{attribute 'qualified_only'}
VAR_GLOBAL
END_VAR

(* stored: Version 1.1.0.1, ProductVersion 3.1.4024.3
   GVL Recipes: Id {25ec8ab5-b8fa-4e44-9a63-9a468b11e98a} *)
